FUNCTION_BLOCK fbSafetyStateAndDiagDecode
VAR_IN_OUT
		SafetyStatus :st_SafetyStatus;
END_VAR
VAR_INPUT 
		State :USINT;
		Diag  :USINT;
END_VAR

SafetyStatus.RawDiagCode:= Diag;
SafetyStatus.RawStateCode:=State;
SafetyStatus.State:=State;
SafetyStatus.FSoEMasterFailSafeActive:=Diag.7;
SafetyStatus.StartUp:= Diag.6;
SafetyStatus.FSoESlaveFailSafeActive:=Diag.5;
SafetyStatus.FSoESlaveError:=Diag.4;
SafetyStatus.Diagnosis:= SHL(Diag,4);

END_FUNCTION_BLOCK

(* stored: Version 1.1.0.1, ProductVersion 3.1.4024.12
   POU fbSafetyStateAndDiagDecode: Id {1bf99c34-53fa-417e-98cb-86241aef3980}, SpecialFunc None *)
